PROGRAM Get_Data
VAR
	fbSqlDatabase	: FB_SQLDatabaseEvt(sNetID := '', tTimeout := T#5S);
	fbSqlCommand	: FB_SQLCommandEvt(sNetID := '', tTimeout := T#5S);
	fbSqlResult		: FB_SQLResultEvt(sNetID:='', tTimeout   := T#5S); 
    
	nState			: INT;
	sCmd			: STRING(1000);
	
	aReadStruct		: ARRAY[1..10] OF ST_SelectStruct;

	count			: LINT;
	lim				: USINT;
	
	exec			: BOOL;
	read			: BOOL;
	rel				: BOOL;
	exec2			: BOOL;
	read2			: BOOL;
	rel2			: BOOL;
END_VAR

IF Main2.done THEN
	nState := 0;
END_IF

(* connect to localdb *)
IF NOT fbSqlDatabase.bConnected THEN
	fbSqlDatabase.Connect(1);
END_IF

IF fbSqlDatabase.bConnected THEN
	
	(* count records *)
	IF nState=0 THEN
		
		fbSqlDatabase.CreateCmd(ADR(fbSqlCommand));
		sCmd := 'SELECT COUNT(*) FROM `buffer_data` ORDER BY datetime ASC';
			
		(* execute query *)
		IF exec:=fbSQLCommand.ExecuteDataReturn(ADR(sCmd), SIZEOF(sCmd), ADR(fbSqlResult)) THEN
			IF fbSQLCommand.bError THEN
				(* execute query error handling *) 
			END_IF
			
			(* read & release cache *)
			read:=fbSqlResult.Read(0, 1, ADR(count), SIZEOF(count), TRUE, TRUE);
			IF rel:=fbSqlResult.Release() THEN
				
				(* determine no of records to select *)
				IF count < 10 THEN
					lim := 1;
				ELSE
					lim := 10;
				END_IF
				
				nState:=1;
			END_IF
		END_IF
		
		
	
	END_IF
	
	(* select records *)
	IF nState = 1 THEN
		
		(* query *)
		sCmd := 'SELECT * FROM `buffer_data` ORDER BY datetime ASC LIMIT ';
		sCmd := CONCAT(sCmd, USINT_TO_STRING(lim));
		
		(* execute query *)
		IF exec2:=fbSQLCommand.ExecuteDataReturn(ADR(sCmd), SIZEOF(sCmd), ADR(fbSqlResult)) THEN
			IF fbSQLCommand.bError THEN
				(* execute query error handling *) 
			END_IF
		END_IF
		
		(* read & release cache *)
		read2:=fbSqlResult.Read(0, lim, ADR(aReadStruct), SIZEOF(aReadStruct), TRUE, TRUE);
		IF rel2:=fbSqlResult.Release() THEN
			nState:=2;
		END_IF
	END_IF
END_IF

END_PROGRAM

(* stored: Version 1.1.0.1, ProductVersion 3.1.4024.6
   POU Get_Data: Id {356e4097-52ca-4291-ab97-d55f16e736e8}, SpecialFunc None *)
